Staubli VAL3: splitString.pgx

public program splitString(string& x_sInput[], string x_sPattern, lists& x_lResult[])
  local num l_nLength
  local num l_nElement
  local string l_sLine
  local num l_nCount
  local num l_nPos
begin

  l_nLength = size(x_sInput)
  resize(x_lResult,1,1)
  resize(x_lResult.sString,1,1)
  x_lResult.sString =""
  resize(x_lResult,1,l_nLength)

  if x_sPattern == ""
    call splitWord(x_sInput, x_lResult)
    return
  else
    // iterate complete input x_sInput[0] ... x_sInput[l_nLength-1]
    for l_nElement = 0 to l_nLength-1

      // copy element
      l_sLine = x_sInput[l_nElement]

      // search x_sPattern
      l_nCount = 0
      while len(l_sLine)!=0
        l_nPos=find(l_sLine, x_sPattern)

        if l_nPos==-1
          l_nPos=len(l_sLine)
        endIf

        if l_nCount != 0
          append(x_lResult[l_nElement].sString)
        endIf

        x_lResult[l_nElement].sString[l_nCount] = left(l_sLine,l_nPos)
        l_sLine = right(l_sLine,max(0,len(l_sLine)-l_nPos-len(x_sPattern)))
        l_nCount = l_nCount+1

      endWhile
    endFor
  endIf
end
